{attribute 'qualified_only'}
{attribute 'strict'}
{attribute 'to_string'}
TYPE NestleProducts :
(
	KitKatChunky := 0,
	KitKat2Bar := 1
);
END_TYPE

(* stored: Version 1.1.0.1
   DUT NestleProducts: Id {731ad174-849a-4b08-8397-325c1fd50b44} *)
